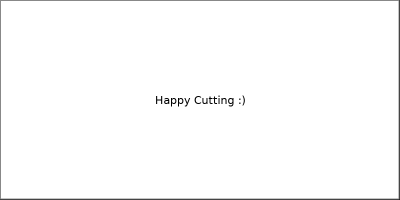
VISUALIZATION V_ProductionNCICircle  // 400x200
VAR_IN_OUT
	HMI : ST_PackMLBaseModule_HMI;
	HMI_GantryXYZ : ST_GantryXYZ_HMI;
	HMI_Recipe : ST_RecipeBuilder_HMI;
END_VAR
    RoundedRectangle (0,0 400x200)
    Label (93,92 215x17), "Happy Cutting :)"
END_VISUALIZATION

(* stored: Version 1.1.0.1, ProductVersion 3.1.4024.15
   Visu V_ProductionNCICircle: Id {4a8c3883-2d70-4998-a8f7-7e4f803d03c4} *)
